// SIMATIC S7-200 SMART project (STEP 7-Micro/WIN SMART), CPU ST60

SYMBOL_TABLE 系统符号
First_Scan_On    SM0.1    // 仅在第一个扫描周期时接通
END_SYMBOL_TABLE

ORGANIZATION_BLOCK MAIN:OB1
TITLE=程序注释
BEGIN
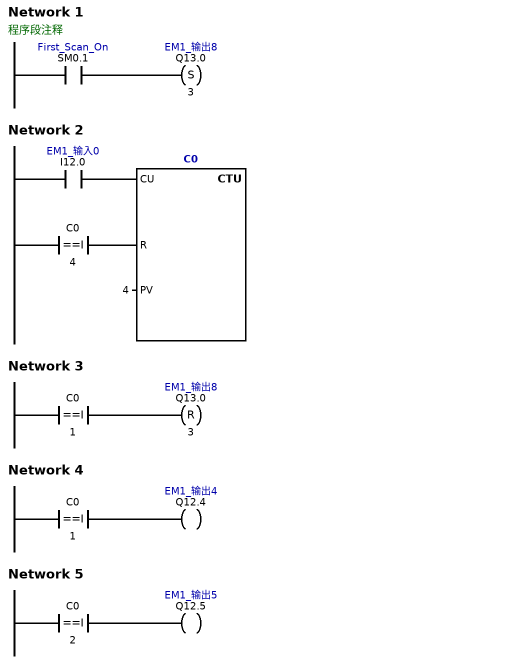
Network 1
// 程序段注释
// (network saved uncompiled; LAD cells follow)
// row 0: c0 -| |- First_Scan_On:SM0.1  c1 -(S) EM1_输出8:Q13.0, 3
Network 2
// (network saved uncompiled; LAD cells follow)
// row 0: c0 -| |- EM1_输入0:I12.0  c1 [CTU C0 CU:=power@row0, R:=power@row1, PV:=4]
// row 1: c0 -|==I|- C0, 4  c1 [box]
// row 2: c1 [box]
Network 3
// (network saved uncompiled; LAD cells follow)
// row 0: c0 -|==I|- C0, 1  c1 -(R) EM1_输出8:Q13.0, 3
Network 4
// (network saved uncompiled; LAD cells follow)
// row 0: c0 -|==I|- C0, 1  c1 -( ) EM1_输出4:Q12.4
Network 5
// (network saved uncompiled; LAD cells follow)
// row 0: c0 -|==I|- C0, 2  c1 -( ) EM1_输出5:Q12.5
END_ORGANIZATION_BLOCK
